FUNCTION SPLIT_WORD_INTO_BYTES (* this Function extracts the 2 BYTE from a word *)
  (* Standard: 61499-1; Description: Copyright (c) 2024 HR Agrartechnik GmbH This program and the accompanying materials are made available under the terms of the Eclipse Public License 2.0 which is available at https://www.eclipse.org/legal/epl-2.0/ SPDX-License-Identifier: EPL-2.0 *)
  (* Version 3.0, 2025-04-14, Patrick Aigner, changed package *)
  (* Version 1.1, 2024-07-24, Moritz Ortmeier, HR Agrartechnik, rename Function and change Output Variables *)
  (* Version 1.0, 2024-02-22, Franz H??pfinger, HR Agrartechnik, initial Implementation *)
  PACKAGE eclipse4diac::utils::splitting;
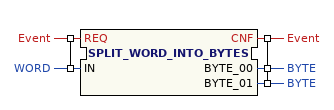
  EVENT_INPUT
    REQ WITH IN; (* Normal Execution Request *)
  END_EVENT
  EVENT_OUTPUT
    CNF WITH BYTE_00, BYTE_01; (* Execution Confirmation *)
  END_EVENT
  VAR_INPUT
    IN : WORD;
  END_VAR
  VAR_OUTPUT
    BYTE_00 : BYTE;
    BYTE_01 : BYTE;
  END_VAR
  BODY IN ST:
(* this Function extracts the 2 BYTE from a word *)
FUNCTION SPLIT_WORD_INTO_BYTES

VAR_INPUT
	IN : WORD;
END_VAR

VAR_OUTPUT
	BYTE_00 : BYTE;
	BYTE_01 : BYTE;
END_VAR

BYTE_00 := IN.%B0;
BYTE_01 := IN.%B1;

END_FUNCTION
  END_BODY
END_FUNCTION
